FUNCTION_BLOCK PV_FILTER (* Basic FB with empty ECC *)
  (* Standard: 61499-2 *)
  (* Version 1.0, 2026-04-29, guilh *)
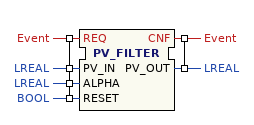
  EVENT_INPUT
    REQ WITH PV_IN, ALPHA, RESET;
  END_EVENT
  EVENT_OUTPUT
    CNF WITH PV_OUT;
  END_EVENT
  VAR_INPUT
    PV_IN : LREAL;
    ALPHA : LREAL;
    RESET : BOOL;
  END_VAR
  VAR_OUTPUT
    PV_OUT : LREAL;
  END_VAR
  VAR
    initialized : BOOL;
    alpha_limited : LREAL;
  END_VAR
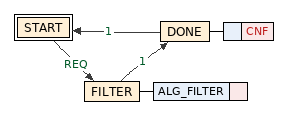
  EC_STATES
    START; (* Initial State *)
    FILTER : ALG_FILTER;
    DONE : -> CNF;
  END_STATES
  EC_TRANSITIONS
    START TO FILTER := REQ;
    FILTER TO DONE := 1;
    DONE TO START := 1;
  END_TRANSITIONS
  ALGORITHM ALG_FILTER IN ST:
IF RESET THEN
    PV_OUT := PV_IN;
    initialized := TRUE;
ELSE
    IF NOT initialized THEN
        PV_OUT := PV_IN;
        initialized := TRUE;
    ELSE
        alpha_limited := ALPHA;

        IF alpha_limited < 0.0 THEN
            alpha_limited := 0.0;
        ELSIF alpha_limited > 1.0 THEN
            alpha_limited := 1.0;
        END_IF;

        PV_OUT := (alpha_limited * PV_OUT) + ((1.0 - alpha_limited) * PV_IN);
    END_IF;
END_IF;
  END_ALGORITHM
END_FUNCTION_BLOCK
